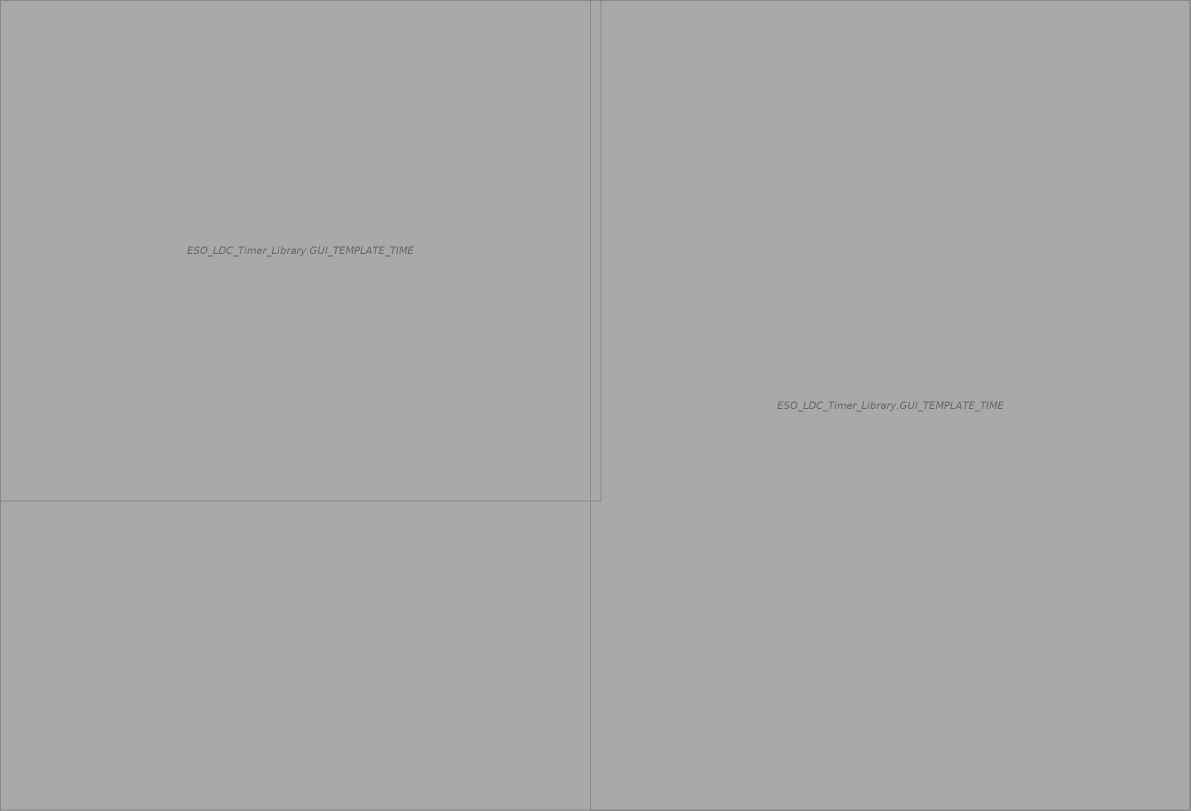
VISUALIZATION VISU_HMI_SERVICES_TIME  // 1191x811
VAR_IN_OUT
	m_Instance : FB_TIME;
    m_Hmi : FB_HMI_SERVICES_TIME;
END_VAR
    Frame (0,0 601x501)
        shows ESO_LDC_Timer_Library.GUI_TEMPLATE_TIME(m_DeviceName := 'time_info', m_Instance := m_Instance)
    Frame (590,0 601x811)
        shows ESO_LDC_Timer_Library.GUI_TEMPLATE_TIME(m_DeviceName := 'time_info', m_Instance := m_Instance)
        p2738717112: m_Hmi.nAbsoluteMovementY
END_VISUALIZATION

(* stored: Version 1.1.0.1, ProductVersion 3.1.4024.14
   Visu VISU_HMI_SERVICES_TIME: Id {f65e2a52-9c0c-4434-84f9-e296b40f771e} *)
